PROGRAM MAIN
VAR
    timer_t: LREAL;
    preset_timer_t: TIME;
    timer: timer_location;
    sup: sup_location;
    hw_button_bit: BOOL;
    hw_button: hw_button_location;
    hw_lamp_bit: BOOL;
    hw_lamp: hw_lamp_location;
    firstRun: BOOL := TRUE;
END_VAR
VAR_TEMP
    curValue: LREAL;
    current_hw_button: hw_button_location;
    current_hw_button_1: hw_button_location;
    current_hw_lamp: hw_lamp_location;
    current_hw_lamp_1: hw_lamp_location;
    current_hw_lamp_bit: BOOL;
    current_hw_lamp_bit_1: BOOL;
    current_sup: sup_location;
    current_sup_1: sup_location;
    current_sup_2: sup_location;
    current_sup_3: sup_location;
    current_sup_4: sup_location;
    current_sup_5: sup_location;
    current_timer: timer_location;
    current_timer_1: timer_location;
    current_timer_t: LREAL;
    eventEnabled: BOOL;
    isProgress: BOOL;
    syncAutEdge: DINT;
    syncAutEdge_1: DINT;
    syncAutEdge_10: DINT;
    syncAutEdge_11: DINT;
    syncAutEdge_2: DINT;
    syncAutEdge_3: DINT;
    syncAutEdge_4: DINT;
    syncAutEdge_5: DINT;
    syncAutEdge_6: DINT;
    syncAutEdge_7: DINT;
    syncAutEdge_8: DINT;
    syncAutEdge_9: DINT;
    timeOut: BOOL;
END_VAR

(* --- Read input from sensors. -------------------------------------------- *)
hw_button_bit := in_hw_button_bit;

(* --- Initialize state or update continuous variables. -------------------- *)
IF firstRun THEN
    firstRun := FALSE;

    (* Initialize the state variables. *)
    timer_t := 0.0;
    (* Reset timer of "timer_t". *)
    preset_timer_t := timer_t;
    ton_timer_t(IN := FALSE, PT := preset_timer_t);
    ton_timer_t(IN := TRUE, PT := preset_timer_t);
    timer := timer_Idle;
    sup := sup_s1;
    hw_button := hw_button_Released;
    hw_lamp_bit := FALSE;
    hw_lamp := hw_lamp_Off;
ELSE
    (* Update remaining time of "timer_t". *)
    ton_timer_t(IN := TRUE, PT := preset_timer_t, Q => timeOut, ET => curValue);
    timer_t := SEL(timeOut, preset_timer_t - curValue, 0.0);
END_IF;

(* --- Process all events. ------------------------------------------------- *)
isProgress := TRUE;
(* Perform events until none can be done anymore. *)
WHILE isProgress DO
    isProgress := FALSE;

    (* Try to perform event "timer.start". *)
    eventEnabled := TRUE;
    IF timer = timer_Idle THEN
        syncAutEdge := 1;
    ELSE
        eventEnabled := FALSE;
    END_IF;
    IF eventEnabled THEN
        IF sup = sup_s3 THEN
            syncAutEdge_1 := 1;
        ELSIF sup = sup_s5 THEN
            syncAutEdge_1 := 2;
        ELSE
            eventEnabled := FALSE;
        END_IF;
    END_IF;
    IF eventEnabled THEN
        isProgress := TRUE;
        current_sup := sup;
        current_timer := timer;
        current_timer_t := timer_t;
        IF syncAutEdge = 1 THEN
            timer_t := 3.0;
            (* Reset timer of "timer_t". *)
            preset_timer_t := timer_t;
            ton_timer_t(IN := FALSE, PT := preset_timer_t);
            ton_timer_t(IN := TRUE, PT := preset_timer_t);
            timer := timer_Running;
        END_IF;
        IF syncAutEdge_1 = 1 THEN
            sup := sup_s6;
        ELSIF syncAutEdge_1 = 2 THEN
            sup := sup_s7;
        END_IF;
    END_IF;

    (* Try to perform event "timer.timeout". *)
    eventEnabled := TRUE;
    IF timer = timer_Running AND timer_t <= 0.0 THEN
        syncAutEdge_2 := 1;
    ELSE
        eventEnabled := FALSE;
    END_IF;
    IF eventEnabled THEN
        IF sup = sup_s6 THEN
            syncAutEdge_3 := 1;
        ELSIF sup = sup_s7 THEN
            syncAutEdge_3 := 2;
        ELSE
            eventEnabled := FALSE;
        END_IF;
    END_IF;
    IF eventEnabled THEN
        isProgress := TRUE;
        current_sup_1 := sup;
        current_timer_1 := timer;
        IF syncAutEdge_2 = 1 THEN
            timer := timer_Idle;
        END_IF;
        IF syncAutEdge_3 = 1 THEN
            sup := sup_s8;
        ELSIF syncAutEdge_3 = 2 THEN
            sup := sup_s9;
        END_IF;
    END_IF;

    (* Try to perform event "button.push". *)
    eventEnabled := TRUE;
    IF sup = sup_s1 THEN
        syncAutEdge_4 := 1;
    ELSIF sup = sup_s4 THEN
        syncAutEdge_4 := 2;
    ELSIF sup = sup_s5 THEN
        syncAutEdge_4 := 3;
    ELSIF sup = sup_s7 THEN
        syncAutEdge_4 := 4;
    ELSIF sup = sup_s9 THEN
        syncAutEdge_4 := 5;
    ELSE
        eventEnabled := FALSE;
    END_IF;
    IF eventEnabled THEN
        IF hw_button = hw_button_Released AND hw_button_bit THEN
            syncAutEdge_5 := 1;
        ELSE
            eventEnabled := FALSE;
        END_IF;
    END_IF;
    IF eventEnabled THEN
        isProgress := TRUE;
        current_hw_button := hw_button;
        current_sup_2 := sup;
        IF syncAutEdge_4 = 1 THEN
            sup := sup_s2;
        ELSIF syncAutEdge_4 = 2 THEN
            sup := sup_s2;
        ELSIF syncAutEdge_4 = 3 THEN
            sup := sup_s3;
        ELSIF syncAutEdge_4 = 4 THEN
            sup := sup_s6;
        ELSIF syncAutEdge_4 = 5 THEN
            sup := sup_s8;
        END_IF;
        IF syncAutEdge_5 = 1 THEN
            hw_button := hw_button_Pushed;
        END_IF;
    END_IF;

    (* Try to perform event "button.release". *)
    eventEnabled := TRUE;
    IF sup = sup_s2 THEN
        syncAutEdge_6 := 1;
    ELSIF sup = sup_s3 THEN
        syncAutEdge_6 := 2;
    ELSIF sup = sup_s6 THEN
        syncAutEdge_6 := 3;
    ELSIF sup = sup_s8 THEN
        syncAutEdge_6 := 4;
    ELSIF sup = sup_s10 THEN
        syncAutEdge_6 := 5;
    ELSE
        eventEnabled := FALSE;
    END_IF;
    IF eventEnabled THEN
        IF hw_button = hw_button_Pushed AND NOT hw_button_bit THEN
            syncAutEdge_7 := 1;
        ELSE
            eventEnabled := FALSE;
        END_IF;
    END_IF;
    IF eventEnabled THEN
        isProgress := TRUE;
        current_hw_button_1 := hw_button;
        current_sup_3 := sup;
        IF syncAutEdge_6 = 1 THEN
            sup := sup_s4;
        ELSIF syncAutEdge_6 = 2 THEN
            sup := sup_s5;
        ELSIF syncAutEdge_6 = 3 THEN
            sup := sup_s7;
        ELSIF syncAutEdge_6 = 4 THEN
            sup := sup_s9;
        ELSIF syncAutEdge_6 = 5 THEN
            sup := sup_s1;
        END_IF;
        IF syncAutEdge_7 = 1 THEN
            hw_button := hw_button_Released;
        END_IF;
    END_IF;

    (* Try to perform event "lamp.on". *)
    eventEnabled := TRUE;
    IF sup = sup_s2 THEN
        syncAutEdge_8 := 1;
    ELSIF sup = sup_s4 THEN
        syncAutEdge_8 := 2;
    ELSE
        eventEnabled := FALSE;
    END_IF;
    IF eventEnabled THEN
        IF hw_lamp = hw_lamp_Off THEN
            syncAutEdge_9 := 1;
        ELSE
            eventEnabled := FALSE;
        END_IF;
    END_IF;
    IF eventEnabled THEN
        isProgress := TRUE;
        current_hw_lamp := hw_lamp;
        current_hw_lamp_bit := hw_lamp_bit;
        current_sup_4 := sup;
        IF syncAutEdge_8 = 1 THEN
            sup := sup_s3;
        ELSIF syncAutEdge_8 = 2 THEN
            sup := sup_s5;
        END_IF;
        IF syncAutEdge_9 = 1 THEN
            hw_lamp_bit := TRUE;
            hw_lamp := hw_lamp_On;
        END_IF;
    END_IF;

    (* Try to perform event "lamp.off". *)
    eventEnabled := TRUE;
    IF sup = sup_s8 THEN
        syncAutEdge_10 := 1;
    ELSIF sup = sup_s9 THEN
        syncAutEdge_10 := 2;
    ELSE
        eventEnabled := FALSE;
    END_IF;
    IF eventEnabled THEN
        IF hw_lamp = hw_lamp_On THEN
            syncAutEdge_11 := 1;
        ELSE
            eventEnabled := FALSE;
        END_IF;
    END_IF;
    IF eventEnabled THEN
        isProgress := TRUE;
        current_hw_lamp_1 := hw_lamp;
        current_hw_lamp_bit_1 := hw_lamp_bit;
        current_sup_5 := sup;
        IF syncAutEdge_10 = 1 THEN
            sup := sup_s10;
        ELSIF syncAutEdge_10 = 2 THEN
            sup := sup_s1;
        END_IF;
        IF syncAutEdge_11 = 1 THEN
            hw_lamp_bit := FALSE;
            hw_lamp := hw_lamp_Off;
        END_IF;
    END_IF;
END_WHILE;

(* --- Write output to actuators. ------------------------------------------ *)
out_hw_lamp_bit := hw_lamp_bit;

END_PROGRAM

(* stored: ProductVersion 3.1.0.18, Version 1.1.0.1 *)
